# EPICS substitutions: db/Beckhoff_3XXX/ecmcEL3751_Scalar.substitutions
file "ecmc_analogInput-chX.template"
{
  pattern {CH_ID, ESLO, EOFF, EGU, PREC}
          {01, "${_ESLO=1}", "${_EOFF=0}", "${_EGU=Raw}", "${_PREC=3}"}
}

file "ecmcEL3751_status-chX.template"
{
  pattern {CH_ID, KEY }
          {01,    "AI"}
}
